{attribute 'qualified_only'}
VAR_GLOBAL
END_VAR

(* stored: Version 1.1.0.1, ProductVersion 3.1.4022.7
   GVL GVL_07_Alarm_Servo_Motor_Robot: Id {8f592e31-6808-4cbb-842e-6918da126fe4} *)
